Fanuc KAREL source: KA00017.KL

PROGRAM KA00017
%NOLOCKGROUP
VAR
  SRC: REAL
  DST: POSITION
BEGIN
  SRC = 2.0
  DST = SRC
END KA00017
